Staubli VAL3: recvRosMsg.pgx

program recvRosMsg(sio& x_sSocket (dimensions=1), Prefix& x_pPrefix (dimensions=1), Header& x_hHeader (dimensions=1), Body& x_bBody (dimensions=1), num& x_nConnFlag (dimensions=1), RosSimpleMsg& x_msg (dimensions=1), bool& x_bValidFlag (dimensions=1))
begin
  // Copyright (c) 2021, Institute for Factory Automation and Production Systems (FAPS)
  //
  // Licensed under the Apache License, Version 2.0 (the "License");
  // you may not use this file except in compliance with the License.
  // You may obtain a copy of the License at
  //
  //     http://www.apache.org/licenses/LICENSE-2.0
  //
  // Unless required by applicable law or agreed to in writing, software
  // distributed under the License is distributed on an "AS IS" BASIS,
  // WITHOUT WARRANTIES OR CONDITIONS OF ANY KIND, either express or implied.
  // See the License for the specific language governing permissions and
  // limitations under the License.


  // attempt to receive the data of the message (prefix and header are in x_msg)
  x_pPrefix.nLength=x_msg.prefix.nLength
  x_hHeader.nMsgType=x_msg.header.nMsgType
  x_hHeader.nCommType=x_msg.header.nCommType
  x_hHeader.nReplyCode=x_msg.header.nReplyCode

  call recvData(x_sSocket,x_bBody.nData,x_nConnFlag,x_bValidFlag)
end
